// TIA Portal V21 export
TYPE "MotorPos_CFG_Type_1"
   STRUCT
      xEncoderReversal { S7_SetPoint := 'True'} : Bool;   // Motor encoder direction inversion 0=straight 1=inversion / Inversione direzione encoder motore 0=diritto 1=inversione
      xLaserPhotEncoder { S7_SetPoint := 'True'} : Bool;   // Fotocellula Laser o Encoder (0=Encoder)
      fEncoderRatio { S7_SetPoint := 'True'} : Real := 1.0;   // Encoder points conversion value -> mm (1 encoder turn=movement mm) / Valore di conversione punti encoder -> mm (1 giro encoder=spostamento mm)
      fJogSpeed { S7_SetPoint := 'True'} : Real := 10.0;   // Speed Jog movement (mm/sec) / Velocità movimentazione in jog/Speed Jog moviment (mm/sec)
      fJogAcc { S7_SetPoint := 'True'} : Real := 10.0;   // Acc. jog movement (mm/sec^2) / Acc. movimentazione in jog/Acc. jog movement (mm/sec^2)
      fJogDec { S7_SetPoint := 'True'} : Real := 10.0;   // Dec. jog movement (mm/sec^2) / Dec. movimentazione in jog/Dec. jog movement (mm/sec^2)
      fVirtEncWindPos { S7_SetPoint := 'True'} : Real := 1.0;   // Cycle end virtual encoder position window (mm) / Finestra di posizione encoder virtuale fine ciclo/Window pos. V. encoder(mm)
      fVirtEncWindSpeed { S7_SetPoint := 'True'} : Real := 10.0;   // Cycle end virtual encoder speed window(mm/sec) / Finestra di velocità encoder virtuale fine ciclo/Window speed V. encod(mm/sec)
      fMotWindPos { S7_SetPoint := 'True'} : Real := 1.0;   // Cycle end motor position window (mm) / Finestra di posizione motore fine ciclo/Window motor pos. end cycle (mm)
      fMotWindSpeed { S7_SetPoint := 'True'} : Real := 10.0;   // Cycle end motor speed window (mm/sec) / Finestra di velocità motore fine ciclo/Window motor speed end cycle (mm/sec)
      fMaxErrEnc { S7_SetPoint := 'True'} : Real := 5.0;   // Max tracking value for alarm (mm) / Massimo valore inseguimento per allarme/Max value pursuit alarm (mm)
      fKPpid_Pos { S7_SetPoint := 'True'} : Real := 1.0;   // PID Proportional constant / Anello Posizione Costante proporzionale PID/Proportionale constant PID
      fKPpidAcc_Pos { S7_SetPoint := 'True'} : Real := 1.0;   // Anello Posizione Costante proporzionale PID fase accelerazione/proprotional constant PID dec.
      fKPpidDec_Pos { S7_SetPoint := 'True'} : Real := 4.0;   // PID Proportional constant dec.phase / Anello Posizione Costante proporzionale PID fase decelerazione/proprotional constant PID dec.
      fKPpid_Vel { S7_SetPoint := 'True'} : Real := 1.0;   // Anello Velocità Costante proporzionale PID/Proportionale constant PID
      fKPpidAcc_Vel { S7_SetPoint := 'True'} : Real := 1.0;   // Anello Velocità Costante proporzionale PID fase accelerazione/proprotional constant PID dec.
      fKPpidDec_Vel { S7_SetPoint := 'True'} : Real := 1.0;   // Anello Velocità Costante proporzionale PID fase decelerazione/proprotional constant PID dec.
      fMinSpeed { S7_SetPoint := 'True'} : Real;   // Low limit speed requested (mm/sec) / Limite basso velocità richiesta/Low limit speed requested (mm/sec)
      fMaxSpeed { S7_SetPoint := 'True'} : Real := 100.0;   // High speed limit (mm/sec) / Limite alto velocità richiesta/High speed limit (mm/sec)
      fFirstStepNepero { S7_SetPoint := 'True'} : Real := 6.0;   // Definisce gardino di ingresso Funzione Nepero
      dnTimerStopEnable { S7_SetPoint := 'True'} : DInt := DINT#300;   // Value timer run inverter request (mS) / Valore timer stop richiesta marcia inverter/Value timer run inveter reques (mS)
      dnTimerStopEndPos { S7_SetPoint := 'True'} : DInt := DINT#1000;   // Value timer alarm positioner / Valore timer allarme controllo fine posizionamento/Value timer alarm positioner
   END_STRUCT;
END_TYPE
